FUNCTION_BLOCK Q_ObjHideShow_AX (* Command Hide/Show Object with AX adapter (BOOL) *)
  (* Standard: 61499-2; Description: Copyright (c) 2026 Meisterschulen am Ostbahnhof This program and the accompanying materials are made available under the terms of the Eclipse Public License 2.0 which is available at https://www.eclipse.org/legal/epl-2.0/ SPDX-License-Identifier: EPL-2.0 *)
  (* Version 1.0, 2026-04-24, Franz Höpfinger, Meisterschulen am Ostbahnhof, AX adapter wrapper for Q_ObjHideShow *)
  PACKAGE isobus::UT::Q;
  IMPORT adapter::types::unidirectional::AX;
  IMPORT isobus::UT::Q::Q_ObjHideShow;
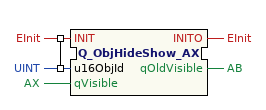
  EVENT_INPUT
    INIT : EInit WITH u16ObjId; (* Service Initialization *)
  END_EVENT
  EVENT_OUTPUT
    INITO : EInit; (* Initialization Confirm *)
  END_EVENT
  VAR_INPUT
    u16ObjId : UINT; (* Object ID *)
  END_VAR
  SOCKETS
    qVisible : adapter::types::unidirectional::AX; (* 0 == hidden, 1 == shown *)
  END_SOCKETS
  PLUGS
    qOldVisible : adapter::types::unidirectional::AB; (* Old value of Visible 0 == hidden, 1 == shown, 0xFF == undefined *)
  END_PLUGS
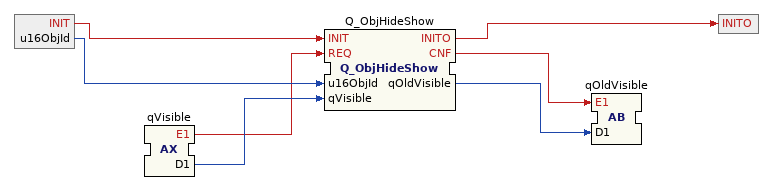
  FBS
    Q_ObjHideShow : isobus::UT::Q::Q_ObjHideShow;
  END_FBS
  EVENT_CONNECTIONS
    INIT TO Q_ObjHideShow.INIT;
    Q_ObjHideShow.INITO TO INITO;
    qVisible.E1 TO Q_ObjHideShow.REQ;
    Q_ObjHideShow.CNF TO qOldVisible.E1;
  END_CONNECTIONS
  DATA_CONNECTIONS
    u16ObjId TO Q_ObjHideShow.u16ObjId;
    qVisible.D1 TO Q_ObjHideShow.qVisible;
    Q_ObjHideShow.qOldVisible TO qOldVisible.D1;
  END_CONNECTIONS
END_FUNCTION_BLOCK
